// Mitsubishi GX Works2 project: 자동 - 복사본   PLC: Q02/Q02H

PROGRAM MAIN
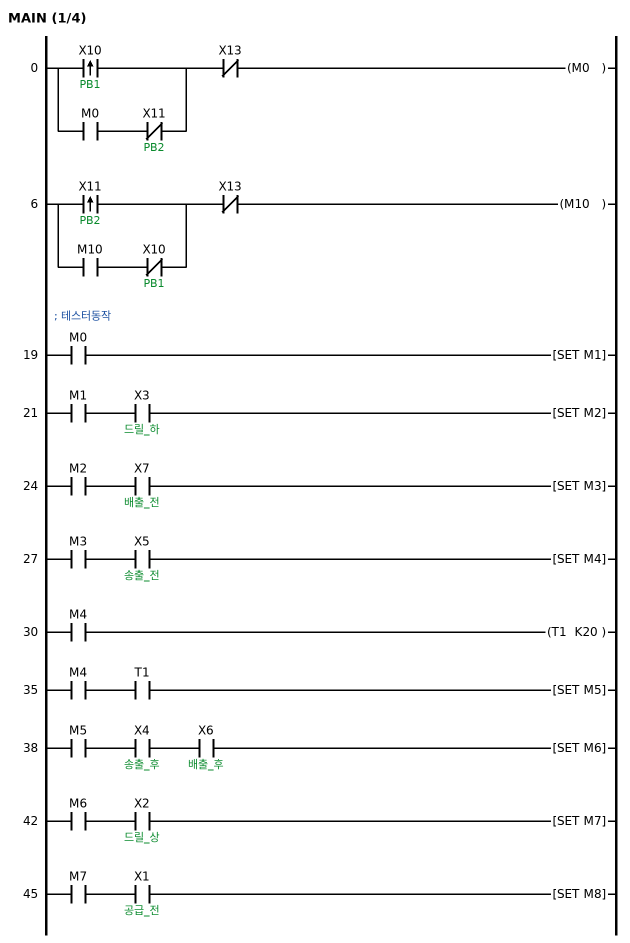
0     LDP     X10  ; PB1
      LD      M0
      ANI     X11  ; PB2
      ORB
      ANI     X13
      OUT     M0
6     LDP     X11  ; PB2
      LD      M10
      ANI     X10  ; PB1
      ORB
      ANI     X13
      OUT     M10
; 테스터동작
19    LD      M0
      SET     M1
21    LD      M1
      AND     X3  ; 드릴_하
      SET     M2
24    LD      M2
      AND     X7  ; 배출_전
      SET     M3
27    LD      M3
      AND     X5  ; 송출_전
      SET     M4
30    LD      M4
      OUT     T1 K20
35    LD      M4
      AND     T1
      SET     M5
38    LD      M5
      AND     X4  ; 송출_후
      AND     X6  ; 배출_후
      SET     M6
42    LD      M6
      AND     X2  ; 드릴_상
      SET     M7
45    LD      M7
      AND     X1  ; 공급_전
      SET     M8
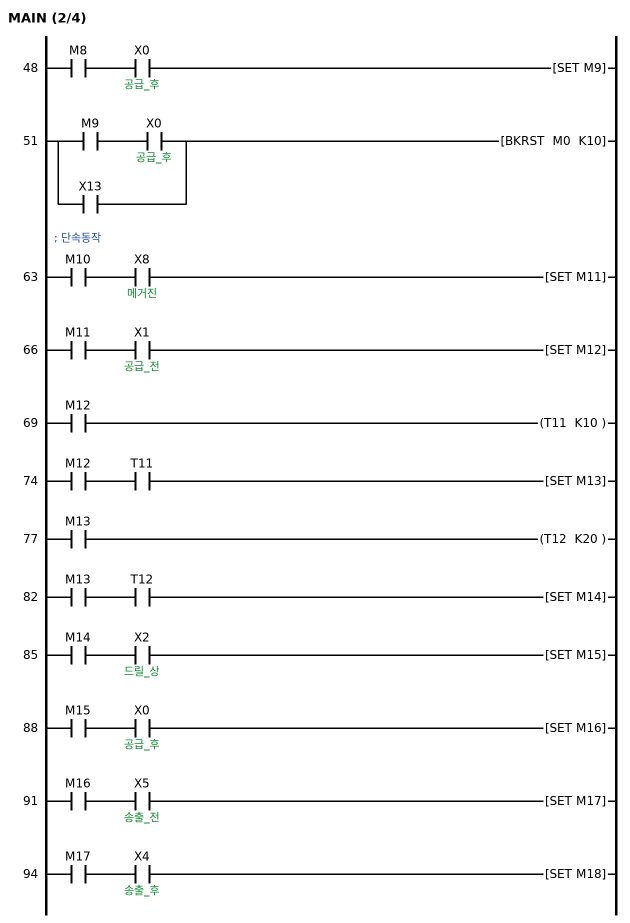
48    LD      M8
      AND     X0  ; 공급_후
      SET     M9
51    LD      M9
      AND     X0  ; 공급_후
      OR      X13
      BKRST   M0 K10
; 단속동작
63    LD      M10
      AND     X8  ; 메거진
      SET     M11
66    LD      M11
      AND     X1  ; 공급_전
      SET     M12
69    LD      M12
      OUT     T11 K10
74    LD      M12
      AND     T11
      SET     M13
77    LD      M13
      OUT     T12 K20
82    LD      M13
      AND     T12
      SET     M14
85    LD      M14
      AND     X2  ; 드릴_상
      SET     M15
88    LD      M15
      AND     X0  ; 공급_후
      SET     M16
91    LD      M16
      AND     X5  ; 송출_전
      SET     M17
94    LD      M17
      AND     X4  ; 송출_후
      SET     M18
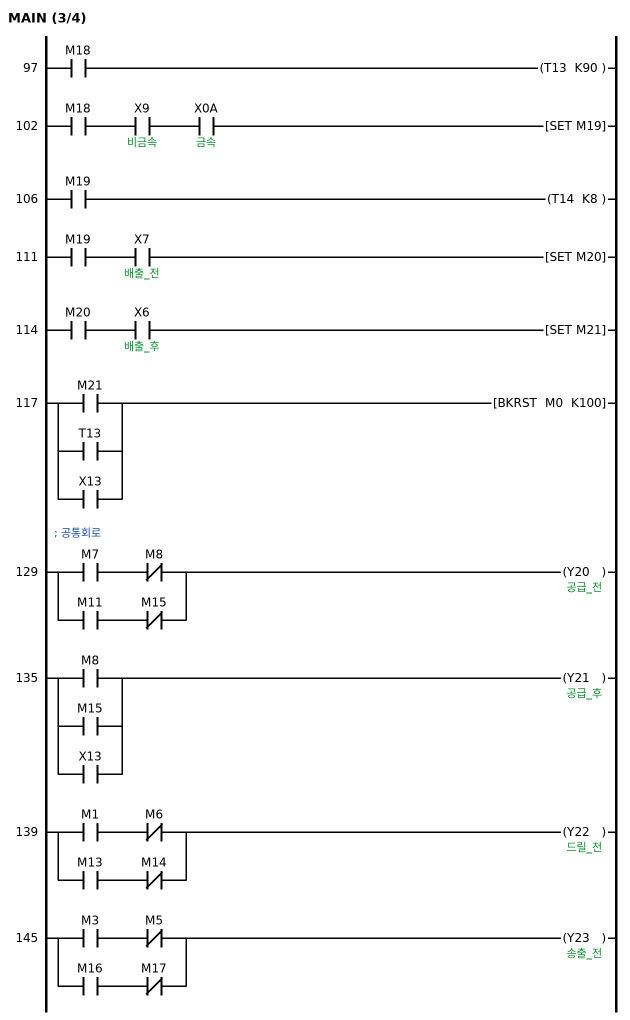
97    LD      M18
      OUT     T13 K90
102   LD      M18
      AND     X9  ; 비금속
      AND     X0A  ; 금속
      SET     M19
106   LD      M19
      OUT     T14 K8
111   LD      M19
      AND     X7  ; 배출_전
      SET     M20
114   LD      M20
      AND     X6  ; 배출_후
      SET     M21
117   LD      M21
      OR      T13
      OR      X13
      BKRST   M0 K100
; 공통회로
129   LD      M7
      ANI     M8
      LD      M11
      ANI     M15
      ORB
      OUT     Y20  ; 공급_전
135   LD      M8
      OR      M15
      OR      X13
      OUT     Y21  ; 공급_후
139   LD      M1
      ANI     M6
      LD      M13
      ANI     M14
      ORB
      OUT     Y22  ; 드릴_전
145   LD      M3
      ANI     M5
      LD      M16
      ANI     M17
      ORB
      OUT     Y23  ; 송출_전
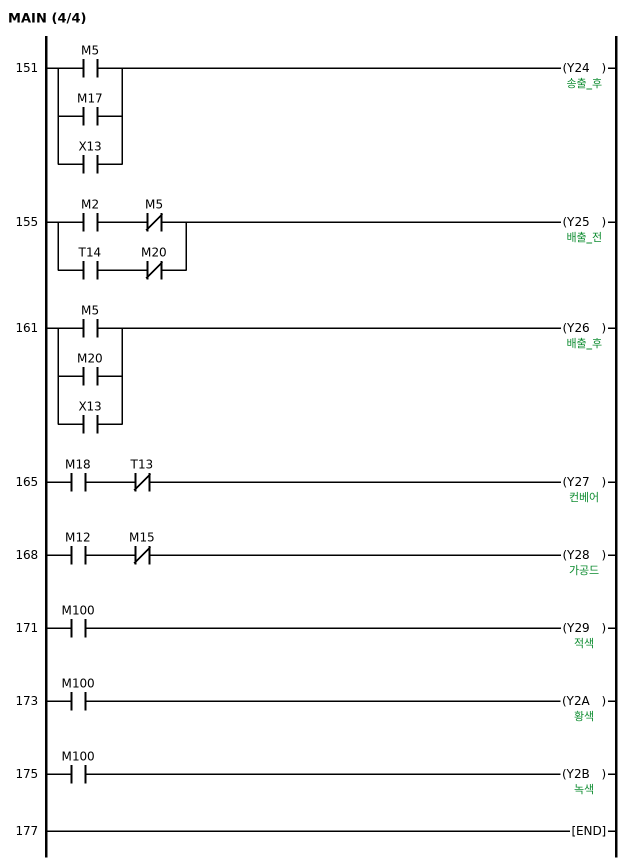
151   LD      M5
      OR      M17
      OR      X13
      OUT     Y24  ; 송출_후
155   LD      M2
      ANI     M5
      LD      T14
      ANI     M20
      ORB
      OUT     Y25  ; 배출_전
161   LD      M5
      OR      M20
      OR      X13
      OUT     Y26  ; 배출_후
165   LD      M18
      ANI     T13
      OUT     Y27  ; 컨베어
168   LD      M12
      ANI     M15
      OUT     Y28  ; 가공드
171   LD      M100
      OUT     Y29  ; 적색
173   LD      M100
      OUT     Y2A  ; 황색
175   LD      M100
      OUT     Y2B  ; 녹색
177   END
END_PROGRAM

PROGRAM MAIN1
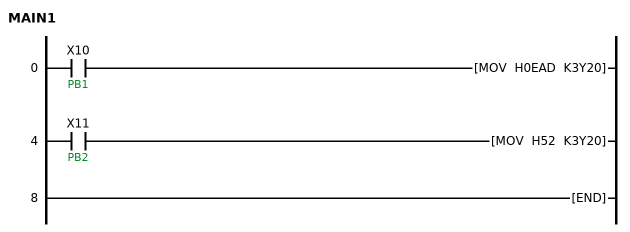
0     LD      X10  ; PB1
      MOV     H0EAD K3Y20  ; 공급_전
4     LD      X11  ; PB2
      MOV     H52 K3Y20
8     END
END_PROGRAM

PROGRAM MAIN2
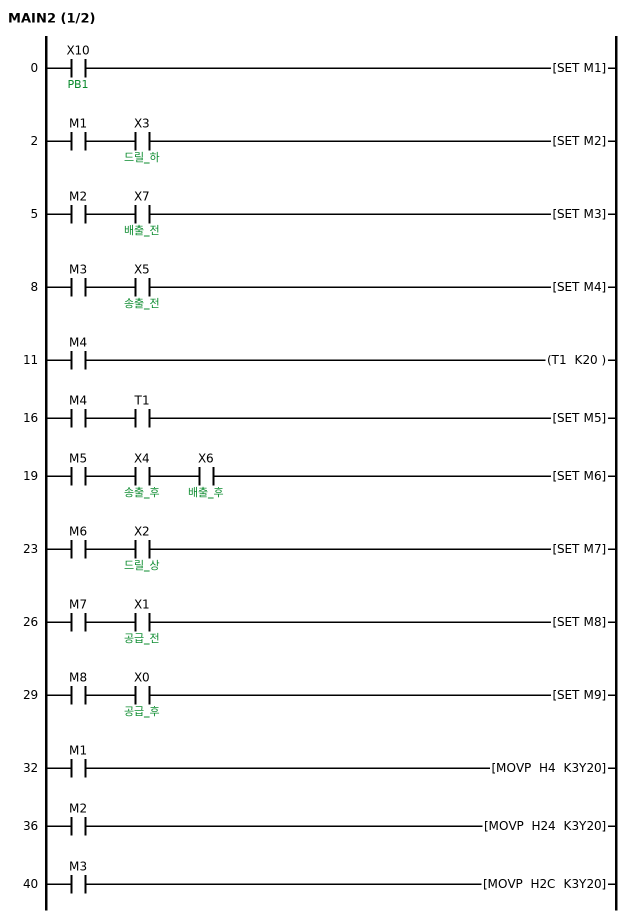
0     LD      X10  ; PB1
      SET     M1
2     LD      M1
      AND     X3  ; 드릴_하
      SET     M2
5     LD      M2
      AND     X7  ; 배출_전
      SET     M3
8     LD      M3
      AND     X5  ; 송출_전
      SET     M4
11    LD      M4
      OUT     T1 K20
16    LD      M4
      AND     T1
      SET     M5
19    LD      M5
      AND     X4  ; 송출_후
      AND     X6  ; 배출_후
      SET     M6
23    LD      M6
      AND     X2  ; 드릴_상
      SET     M7
26    LD      M7
      AND     X1  ; 공급_전
      SET     M8
29    LD      M8
      AND     X0  ; 공급_후
      SET     M9
32    LD      M1
      MOVP    H4 K3Y20  ; 공급_전
36    LD      M2
      MOVP    H24 K3Y20
40    LD      M3
      MOVP    H2C K3Y20
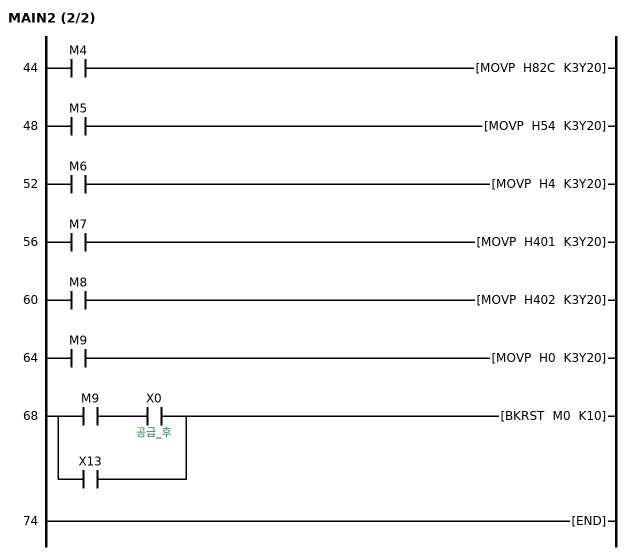
44    LD      M4
      MOVP    H82C K3Y20
48    LD      M5
      MOVP    H54 K3Y20
52    LD      M6
      MOVP    H4 K3Y20
56    LD      M7
      MOVP    H401 K3Y20
60    LD      M8
      MOVP    H402 K3Y20
64    LD      M9
      MOVP    H0 K3Y20
68    LD      M9
      AND     X0  ; 공급_후
      OR      X13
      BKRST   M0 K10
74    END
END_PROGRAM

// device comments not shown above
X12  ; PB3
